// TIA Portal V17 export
// export: Created 2023-09-09T00:07:24.0498182Z, ExportSetting WithDefaults, DisplayName Totally Integrated Automation Portal, DisplayVersion V17 Update 6, DisplayName TIA Portal Openness, DisplayVersion V17 Update 6, DisplayName TIA Portal Teamcenter Gateway, DisplayVersion V17 Update 6, DisplayName TIA Portal Version Control Interface, DisplayVersion V17, DisplayName Simotion SCOUT TIA, DisplayVersion 5.4.3.0, DisplayName TIA Portal Test Suite Advanced, DisplayVersion V17 Update 1, DisplayName SIMOCODE ES, DisplayVersion V17 Update 5, DisplayName SINAMICS Startdrive Advanced, DisplayVersion V17 SP1, DisplayName SINAMICS Startdrive G130, G150, S120, S150, SINAMICS MV, S210, DisplayVersion V17 SP1, DisplayName SINAMICS Startdrive G110M, G120, G120C, G120D, G120P, G115D, DisplayVersion V17 SP1, DisplayName SIRIUS Safety ES, DisplayVersion V17 Update 5, DisplayName STEP 7 Professional, DisplayVersion V17 Update 6, DisplayName STEP 7 CFC, DisplayVersion V17 Update 1, DisplayName STEP 7 Safety, DisplayVersion V17 Update 6, DisplayName WinCC Advanced, DisplayVersion V17 Update 6, DisplayName SIMATIC Visualization Architect, DisplayVersion V17 Update 5
DATA_BLOCK "02_COM"   // DB4, F_DB
{ S7_Optimized_Access := 'TRUE' }
VERSION : 0.1
// stored: AutoNumber true, DBAccessibleFromOPCUA true, DBAccessibleFromWebserver true
   VAR
      EXAMPLE_SORTER_PB : Bool;
      EXAMPLE_SORTER_FDB { ExternalWritable := 'False'} : Bool;
      EXAMPLE_ZONE3_PB { ExternalWritable := 'False'} : Bool;
      EXAMPLE_ZONE3_FDB { ExternalWritable := 'False'} : Bool;
      S1_PB : Bool := False;   // ^SORTER UPPER COY =SC01
      S1_FDB : Bool := False;   // ^SORTER UPPER COY =SC01
      S2_PB : Bool := False;   // ^SORTER LOWER COY =SC02
      S2_FDB : Bool := False;   // ^SORTER LOWER COY =SC02
      S3_PB : Bool := False;   // ^SORTER UPPER FLY =SF03
      S3_FDB : Bool := False;   // ^SORTER UPPER FLY =SF03
      S4_PB : Bool := False;   // ^SORTER LOWER FLY =SF04
      S4_FDB : Bool := False;   // ^SORTER LOWER FLY =SF04
      A1_PB : Bool := False;   // >AREA 1 - INTRO+UPSTREAM COY WEST
      A1_FDB : Bool := False;   // >AREA 1 - INTRO+UPSTREAM COY WEST
      A2_PB : Bool := False;   // >AREA 2 - UPSTREAM FLY WEST 5FSN_115/117
      A2_FDB : Bool := False;   // >AREA 2 - UPSTREAM FLY WEST 5FSN_115/117
      A3_PB : Bool := False;   // >AREA 3 - DOWNSTREAM 5FSN_122
      A3_FDB : Bool := False;   // >AREA 3 - DOWNSTREAM 5FSN_122
      A4_PB : Bool := False;   // >AREA 4 - INTRO+UPSTREAM FLY
      A4_FDB : Bool := False;   // >AREA 4 - INTRO+UPSTREAM FLY
      A5_PB : Bool := False;   // >AREA 5 - INTRO+UPSTREAM COY EAST
      A5_FDB : Bool := False;   // >AREA 5 - INTRO+UPSTREAM COY EAST
      A6_PB : Bool := False;   // >AREA 6 - AREA WEST OF OOG SYSTEM + CALJAN TELESCOPICs + MPSs
      A6_FDB : Bool := False;   // >AREA 6 - AREA WEST OF OOG SYSTEM + CALJAN TELESCOPICs + MPSs
      A7_PB : Bool := False;   // >AREA 7 - AREA EAST OF OOG SYSTEM + CALJAN TELESCOPICs + MPSs
      A7_FDB : Bool := False;   // >AREA 7 - AREA EAST OF OOG SYSTEM + CALJAN TELESCOPICs + MPSs
      L1_PB : Bool := False;   // ~Local C&E: VERTICAL SWITCH UC114 - DOOR: I.2172.3 | =SC00+UC114.VS019-8AF3
      L1_FDB : Bool := False;   // ~Local C&E: VERTICAL SWITCH UC114 - DOOR: I.2172.3 | =SC00+UC114.VS019-8AF3
      L2_PB : Bool := False;   // ~Local C&E: VERTICAL SWITCH UC124 - DOOR: I.2172.3 | =SC00+UC114.VS019-8AF3
      L2_FDB : Bool := False;   // ~Local C&E: VERTICAL SWITCH UC124 - DOOR: I.2172.3 | =SC00+UC114.VS019-8AF3
      L3_PB : Bool := False;   // ~Local C&E: VERTICAL SWITCH UC134 - DOOR: I.2172.3 | =SC00+UC114.VS019-8AF3
      L3_FDB : Bool := False;   // ~Local C&E: VERTICAL SWITCH UC134 - DOOR: I.2172.3 | =SC00+UC114.VS019-8AF3
      L4_PB : Bool := False;   // ~Local C&E: VERTICAL SWITCH UC144 - DOOR: I.2172.3 | =SC00+UC114.VS019-8AF3
      L4_FDB : Bool := False;   // ~Local C&E: VERTICAL SWITCH UC144 - DOOR: I.2172.3 | =SC00+UC114.VS019-8AF3
      L5_PB : Bool := False;   // ~Local C&E: VERTICAL SWITCH UC154 - DOOR: I.2172.3 | =SC00+UC114.VS019-8AF3
      L5_FDB : Bool := False;   // ~Local C&E: VERTICAL SWITCH UC154 - DOOR: I.2172.3 | =SC00+UC114.VS019-8AF3
      L6_PB : Bool := False;   // ~Local C&E: VERTICAL SWITCH UC164 - DOOR: I.2172.3 | =SC00+UC114.VS019-8AF3
      L6_FDB : Bool := False;   // ~Local C&E: VERTICAL SWITCH UC164 - DOOR: I.2172.3 | =SC00+UC114.VS019-8AF3
      L7_PB : Bool := False;   // ~Local C&E: VERTICAL SWITCH UC175 - DOOR: I.2172.3 | =SC00+UC114.VS019-8AF3
      L7_FDB : Bool := False;   // ~Local C&E: VERTICAL SWITCH UC175 - DOOR: I.2172.3 | =SC00+UC114.VS019-8AF3
      L8_PB : Bool := False;   // ~Local C&E: VERTICAL SWITCH UC214 - DOOR: I.2172.3 | =SC00+UC114.VS019-8AF3
      L8_FDB : Bool := False;   // ~Local C&E: VERTICAL SWITCH UC214 - DOOR: I.2172.3 | =SC00+UC114.VS019-8AF3
      L9_PB : Bool := False;   // ~Local C&E: VERTICAL SWITCH UC224 - DOOR: I.2172.3 | =SC00+UC114.VS019-8AF3
      L9_FDB : Bool := False;   // ~Local C&E: VERTICAL SWITCH UC224 - DOOR: I.2172.3 | =SC00+UC114.VS019-8AF3
      L10_PB : Bool := False;   // ~Local C&E: VERTICAL SWITCH UC234 - DOOR: I.2172.3 | =SC00+UC114.VS019-8AF3
      L10_FDB : Bool := False;   // ~Local C&E: VERTICAL SWITCH UC234 - DOOR: I.2172.3 | =SC00+UC114.VS019-8AF3
      L11_PB : Bool := False;   // ~Local C&E: VERTICAL SWITCH UC244 - DOOR: I.2172.3 | =SC00+UC114.VS019-8AF3
      L11_FDB : Bool := False;   // ~Local C&E: VERTICAL SWITCH UC244 - DOOR: I.2172.3 | =SC00+UC114.VS019-8AF3
      L12_PB : Bool := False;   // ~Local C&E: VERTICAL SWITCH UC254 - DOOR: I.2172.3 | =SC00+UC114.VS019-8AF3
      L12_FDB : Bool := False;   // ~Local C&E: VERTICAL SWITCH UC254 - DOOR: I.2172.3 | =SC00+UC114.VS019-8AF3
      L13_PB : Bool := False;   // ~Local C&E: VERTICAL SWITCH UC264 - DOOR: I.2172.3 | =SC00+UC114.VS019-8AF3
      L13_FDB : Bool := False;   // ~Local C&E: VERTICAL SWITCH UC264 - DOOR: I.2172.3 | =SC00+UC114.VS019-8AF3
      L14_PB : Bool := False;   // ~Local C&E: VERTICAL SWITCH UC273 - DOOR: I.2172.3 | =SC00+UC114.VS019-8AF3
      L14_FDB : Bool := False;   // ~Local C&E: VERTICAL SWITCH UC273 - DOOR: I.2172.3 | =SC00+UC114.VS019-8AF3
      L15_PB : Bool := False;   // ~Local C&E: VERTICAL SWITCH UC511 - DOOR: I.2172.3 | =SC00+UC114.VS019-8AF3
      L15_FDB : Bool := False;   // ~Local C&E: VERTICAL SWITCH UC511 - DOOR: I.2172.3 | =SC00+UC114.VS019-8AF3
   END_VAR
BEGIN
END_DATA_BLOCK
